PROGRAM POU
VAR
	
	machine : Machine;
	
	upButton : BOOL := FALSE;
	downButton : BOOL := FALSE;
	
	direction : BOOL := FALSE;
	run : BOOL := TRUE;

END_VAR
VAR // added by the converter: edge detectors and wires of the graphical bodies
    _w1, _w2, _w3, _w4 : BOOL;
END_VAR

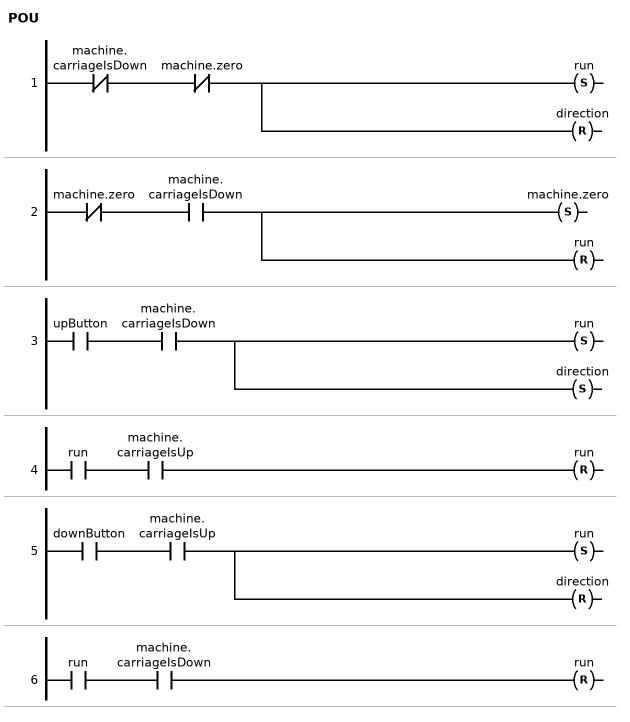
// NETWORK 1
_w1 := NOT machine.carriageIsDown AND NOT machine.zero;
run S= _w1;
direction R= _w1;

// NETWORK 2
_w2 := NOT machine.zero AND machine.carriageIsDown;
machine.zero S= _w2;
run R= _w2;

// NETWORK 3
_w3 := upButton AND machine.carriageIsDown;
run S= _w3;
direction S= _w3;

// NETWORK 4
run R= run AND machine.carriageIsUp;

// NETWORK 5
_w4 := downButton AND machine.carriageIsUp;
run S= _w4;
direction R= _w4;

// NETWORK 6
run R= run AND machine.carriageIsDown;

END_PROGRAM

(* stored: Version 1.1.0.1, ProductVersion 3.1.4024.3
   POU POU: Id {40b0b1dd-6651-4a4c-b59e-54d37f70d1e4}, SpecialFunc None *)
